RoboDK station: Proyecto-Final.rdk

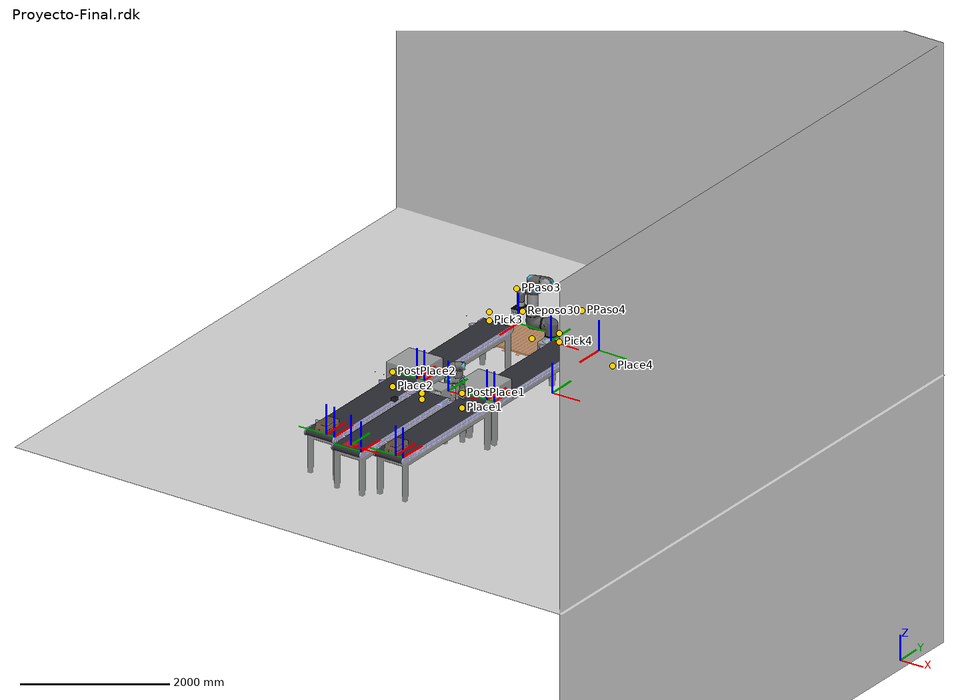
[picture v0: the station drawn from its stored meshes, robots at their saved joint values, targets as dots, program paths as lines]
Station Proyecto final (saved by RoboDK 6.0.0). Poses are relative to the parent item; angles as X-Y-Z fixed-axis rotations.
Station parameters (name, value as stored): SenyalSensor1, 1, SenyalSensor2, 1, SenyalSensorA, 0, SenyalSensor3, 0, SenyalSensor4, 0, x1, 0, z1, 1, x2, 0, z2, 0, x3, 1.0, y3, 0.0, z3, 0.0, x4, 1.0, y4, 0.0, z4, 0.0, Done1, 0, Done2, 0, LuzPalet1, 0, LuzPalet2, 0, IDAzulejo, 23, Lote1, 1, Lote2, 2, ColaAzulejos, 1, Box-Spawner-Settings-4, Box-Spawner-Settings-4-Backup, Box-Spawner-Settings-0, Box-Spawner-Settings-0-Backup, Box-Spawner-Settings-1, Box-Spawner-Settings-1-Backup
  - frame general at (0, -573.6, 0) mm
    - object Wall1 at (3270, -50, -100) mm, rotated rx 0 ry 90 rz 0 deg, size 8910 x 8910 x 0 mm, geometry from Floor.sld
    - object Wall2 at (-1170, 4410, -100) mm, rotated rx 0 ry 90 rz -90 deg, size 8910 x 8910 x 0 mm, geometry from Floor.sld
    - frame UR5e Base at (-1166.19, -738.6, 0) mm
      - robot UR5e: 6 axes, payload 5 kg, reach 850 mm, repeatability 0.03 mm, weight 18.4 kg
          modified DH rows (alpha deg, a mm, theta deg, d mm): 0, 0, 0, 162.5; 90, 0, 180, 0; 0, 425, 0, 0; 0, 392.25, 0, 133.3; -90, 0, 0, 99.7; 90, 0, 180, 99.6
          joint limits [-360, -360, -360, -360, -360, -360] to [360, 360, 360, 360, 360, 360]; home [0, -90, -90, 0, 90, 0]; saved at [128.528, -52.006, 56.851, -94.846, 269.999, -51.472]
        - tool SMC ZXP7A01-ZP20U-X1 Vacuum Gripper, TCP at (0, 0, 125) mm, size 88 x 106.8 x 127.9 mm
    - frame UR30 Base at (-1166.19, 1647.35, -216.33) mm
      - robot UR30: 6 axes
          modified DH rows (alpha deg, a mm, theta deg, d mm): 0, 0, 0, 236.3; 90, 0, 180, 0; 0, 637, 0, 0; 0, 503.7, 0, 201; -90, 0, 0, 159.3; 90, 0, 180, 150
          joint limits [-360, -360, -360, -360, -360, -360] to [360, 360, 360, 360, 360, 360]; home [0, -90, -90, 0, 90, 0]; saved at [-73.932, -91.682, -77.512, -100.814, -269.956, 16.068]
        - tool OnRobot VGP20 Vacuum Gripper, TCP at (-28.8, 0, 85.19) mm, size 214.7 x 147.3 x 83 mm
    - frame Cinta1 at (-372.38, -2930, 100) mm, rotated rx 0 ry 0 rz 90 deg
      - robot Cajas1: 1 axes
          modified DH rows (alpha deg, a mm, theta deg, d mm): 0, 0, 0, 0 linear
          base shift (0, 0, 0) mm, rotated rx 0 ry 90 rz 0 deg
          joint limits [-500000] to [500000]; home [0]; saved at [0]
        - frame CintaCaja1 at (0, 120, 0) mm
          - object cajaA1 at (0, 0, 0) mm, size 193.3 x 289.9 x 121.2 mm, geometry from Box-24x16in-Open.sld
      - object Fotocelula1 at (1900, 0, 0) mm, rotated rx 90 ry 0 rz 90 deg, size 683.3 x 45.2 x 12.5 mm, geometry from SICK-WL4S-Laser-Sensor.sld
      - target Place1 (Cartesian target) at (1686, 221, 9.7) mm, rotated rx -180 ry 0 rz -180 deg; joints [128.527, -47.564, 68.767, -111.204, 269.999, -51.473] of UR5e
      - target PostPlace1 (Cartesian target) at (1686, 221, 226.03) mm, rotated rx 180 ry 0 rz 180 deg; joints [128.527, -51.577, 43.492, -81.916, 269.999, -51.473] of UR5e
    - frame Cinta2 at (-1498.56, -2930, 100) mm, rotated rx 0 ry 0 rz 90 deg
      - robot Cajas2: 1 axes
          modified DH rows (alpha deg, a mm, theta deg, d mm): 0, 0, 0, 0 linear
          base shift (0, 0, 0) mm, rotated rx 0 ry 90 rz 0 deg
          joint limits [-500000] to [500000]; home [0]; saved at [0]
        - frame CintaCaja2 at (0, 120, 0) mm
          - object cajaA2 at (0, 0, 0) mm, size 193.3 x 289.9 x 121.2 mm, geometry from Box-24x16in-Open.sld
      - object Fotocelula2 at (1900, 0, 0) mm, rotated rx 90 ry 0 rz 90 deg, size 683.3 x 45.2 x 12.5 mm, geometry from SICK-WL4S-Laser-Sensor.sld
      - target Place2 (Cartesian target) at (1686, 221, 9.7) mm, rotated rx 180 ry 0 rz 180 deg; joints [32.16, -49.513, 72.223, -112.711, 270.001, -147.84] of UR5e
      - target PostPlace2 (Cartesian target) at (1686, 221, 226.03) mm, rotated rx 180 ry 0 rz 180 deg; joints [32.16, -54.32, 48.04, -83.72, 270.001, -147.84] of UR5e
    - frame Azulejos at (-940.42, -3100.32, 100) mm, rotated rx 0 ry 0 rz 90 deg
      - robot AzulejoAn: 1 axes
          modified DH rows (alpha deg, a mm, theta deg, d mm): 0, 0, 0, 0 linear
          base shift (0, 0, 0) mm, rotated rx 0 ry 90 rz 0 deg
          joint limits [-500000] to [500000]; home [0]; saved at [0]
        - frame CintaAzulejos at (90, 230, 0) mm, rotated rx 0 ry 0 rz -90 deg
          - object Azulejo at (0, 0, 0) mm, size 176.4 x 137.2 x 9.8 mm, geometry from tinker.obj
          - object Azulejo at (0, 0, 0) mm, size 176.4 x 137.2 x 9.8 mm, geometry from tinker.obj
          - object Azulejo at (0, 0, 0) mm, size 176.4 x 137.2 x 9.8 mm, geometry from tinker.obj
          - object Azulejo at (0, 0, 0) mm, size 176.4 x 137.2 x 9.8 mm, geometry from tinker.obj
          - object Azulejo at (0, 0, 0) mm, size 176.4 x 137.2 x 9.8 mm, geometry from tinker.obj
          - object Azulejo at (0, 0, 0) mm, size 176.4 x 137.2 x 9.8 mm, geometry from tinker.obj
          - object Azulejo at (0, 0, 0) mm, size 176.4 x 137.2 x 9.8 mm, geometry from tinker.obj
          - object Azulejo at (0, 0, 0) mm, size 176.4 x 137.2 x 9.8 mm, geometry from tinker.obj
          - object Azulejo at (0, 0, 0) mm, size 176.4 x 137.2 x 9.8 mm, geometry from tinker.obj
          - object Azulejo at (0, 0, 0) mm, size 176.4 x 137.2 x 9.8 mm, geometry from tinker.obj
          - object Azulejo at (0, 0, 0) mm, size 176.4 x 137.2 x 9.8 mm, geometry from tinker.obj
      - object Matrox Iris GTR Camera at (1130, 180, 310) mm, rotated rx 180 ry 0 rz 180 deg, size 76.3 x 92.1 x 55 mm, geometry from Matrox-Iris-GTR-Camera.sld
      - object FotocelulaA at (1850, 0, 0) mm, rotated rx 0 ry 0 rz 90 deg, size 683.3 x 45.2 x 12.5 mm, geometry from SICK-WL4S-Laser-Sensor.sld
      - target Pick (Cartesian target) at (1766.53, 242.5, 8) mm, rotated rx 180 ry 0 rz 180 deg; joints [75.453, -68.071, 102.923, -124.853, 270, -104.547] of UR5e
      - target PrePick (Cartesian target) at (1766.53, 242.5, 95) mm, rotated rx 180 ry 0 rz 180 deg; joints [75.453, -73.796, 96.44, -112.645, 270, -104.547] of UR5e
    - frame Cinta3 at (-1498.56, -835, 100) mm, rotated rx 0 ry 0 rz 90 deg
      - robot Cajas3: 1 axes
          modified DH rows (alpha deg, a mm, theta deg, d mm): 0, 0, 0, 0 linear
          base shift (0, 0, 0) mm, rotated rx 0 ry 90 rz 0 deg
          joint limits [-500000] to [500000]; home [0]; saved at [0]
        - frame CintaCaja3 at (0, 120, 0) mm
          - object cajaC at (0, 0, 0) mm, size 181.1 x 277.6 x 121.7 mm, geometry from Box-24x16in-Closed.sld
          - object cajaC at (0, 0, 0) mm, size 181.1 x 277.6 x 121.7 mm, geometry from Box-24x16in-Closed.sld
      - object Fotocelula3 at (1900, 0, 0) mm, rotated rx 90 ry 0 rz 90 deg, size 683.3 x 45.2 x 12.5 mm, geometry from SICK-WL4S-Laser-Sensor.sld
      - target Pick3 (Cartesian target) at (1780.34, 185.56, 120.53) mm, rotated rx 179.98 ry 0.04 rz 90 deg; joints [-114.864, -111.118, -87.209, -71.708, -269.972, -24.864] of UR30
      - target PrePick3 (Cartesian target) at (1780.34, 185.56, 250.53) mm, rotated rx 179.98 ry 0.04 rz 90 deg; joints [-114.864, -108.804, -75.427, -85.804, -269.972, -24.864] of UR30
    - frame Cinta4 at (-352.38, -835, 100) mm, rotated rx 0 ry 0 rz 90 deg
      - robot Cajas4: 1 axes
          modified DH rows (alpha deg, a mm, theta deg, d mm): 0, 0, 0, 0 linear
          base shift (0, 0, 0) mm, rotated rx 0 ry 90 rz 0 deg
          joint limits [-500000] to [500000]; home [0]; saved at [0]
        - frame CintaCaja4 at (0, 120, 0) mm
          - object cajaC at (0, 0, 0) mm, size 181.1 x 277.6 x 121.7 mm, geometry from Box-24x16in-Closed.sld
          - object cajaC at (0, 0, 0) mm, size 181.1 x 277.6 x 121.7 mm, geometry from Box-24x16in-Closed.sld
      - object Fotocelula4 at (1900, 0, 0) mm, rotated rx 90 ry 0 rz 90 deg, size 683.3 x 45.2 x 12.5 mm, geometry from SICK-WL4S-Laser-Sensor.sld
      - target Pick4 (Cartesian target) at (1780.34, 191.73, 121.32) mm, rotated rx 179.98 ry 0.04 rz 90 deg; joints [-37.962, -112.539, -85.01, -72.432, -269.96, 52.038] of UR30
      - target PrePick4 (Cartesian target) at (1780.34, 191.73, 250.53) mm, rotated rx 179.98 ry 0.04 rz 90 deg; joints [-37.962, -110.369, -73.215, -86.397, -269.96, 52.038] of UR30
    - frame Frame Pallet 1 at (-2170, 2320, -500) mm, rotated rx 0 ry 0 rz -90 deg
      - object Pallet 1130x1130mm at (0, 0, 0) mm, size 706 x 706 x 68.7 mm, geometry from Pallet-1130x1130mm.sld
      - target PPaso3 (Cartesian target) at (739.69, 485.83, 940.76) mm, rotated rx 179.98 ry 0.04 rz -90 deg; joints [-151.611, -76.512, -99.315, -94.218, -269.999, -61.611] of UR30
      - target Place3 (Cartesian target) at (489, 561.4, 120.9) mm, rotated rx 179.98 ry 0.04 rz -90 deg; joints [-177.865, -156.304, -147.246, 33.509, -270.018, -87.865] of UR30
    - frame Frame Pallet 2 at (-812, 2253.67, -500) mm, rotated rx 0 ry 0 rz -90 deg
      - object Pallet 1130x1130mm at (0, 0, 0) mm, size 706 x 706 x 68.7 mm, geometry from Pallet-1130x1130mm.sld
      - target PPaso4 (Cartesian target) at (753.36, 247.81, 965.73) mm, rotated rx 179.98 ry 0.04 rz -90 deg; joints [5.462, -80.617, -93.419, -95.922, -269.984, 95.462] of UR30
      - target Place4 (Cartesian target) at (489, 561.4, 120.9) mm, rotated rx 179.98 ry 0.04 rz -90 deg; joints [-177.865, -156.304, -147.246, 33.509, -270.018, -87.865] of UR30
    - object Mesa4 at (-590, 170, -580) mm, size 465.3 x 1980 x 594 mm, geometry from tinker.obj
    - object Mesa1 at (-590, -1910, -580) mm, size 465.3 x 1980 x 594 mm, geometry from tinker.obj
    - object Mesa2 at (-1720, -1910, -580) mm, size 465.3 x 1980 x 594 mm, geometry from tinker.obj
    - object Mesa3 at (-1720, 170, -580) mm, size 465.3 x 1980 x 594 mm, geometry from tinker.obj
    - object MesaA at (-1160, -2090, -580) mm, size 465.3 x 1980 x 594 mm, geometry from tinker.obj
    - object Soporte30 at (-1166.19, 1647.35, -576.33) mm, size 270 x 270 x 360 mm, geometry from tinker.obj
    - object Soporte5e at (-1166.19, -738.6, -575) mm, size 225 x 225 x 576 mm, geometry from tinker.obj
    - object Tapa1 at (-592, -750, 70) mm, rotated rx 0 ry 0 rz 90 deg, size 540 x 540 x 243 mm, geometry from tinker.obj
    - object Tapa2 at (-1718, -750, 70) mm, rotated rx 0 ry 0 rz 90 deg, size 540 x 540 x 243 mm, geometry from tinker.obj
    - object Basura at (-1158, -950, 60) mm, rotated rx 0 ry 0 rz 90 deg, size 218.7 x 218.7 x 98.4 mm, geometry from tinker.obj
      - object BasuraBajo at (0, 0, 50) mm, rotated rx 180 ry 0 rz 180 deg, size 218.7 x 218.7 x 98.4 mm, geometry from tinker.obj
    - object Floor at (-1140, -50, -570) mm, size 8910 x 8910 x 0 mm, geometry from Floor.sld
    - target Reposo30 (Cartesian target) at (-1144.17, 945.31, 515.93) mm, rotated rx 179.98 ry 0.04 rz 180 deg; joints [-71.585, -90.912, -88.057, -91.037, -269.956, 18.415] of UR30
    - target PuntoPaso1 (Cartesian target) at (-1097.88, -1258.79, 521.04) mm, rotated rx 180 ry 0 rz -90 deg; joints [82.762, -83.23, 58.981, -65.751, 270, -97.238] of UR5e
  - object AzulejoBase at (0, 0, 0) mm, size 176.4 x 137.2 x 9.8 mm, geometry from tinker.obj
  - object cajaBase at (0, 0, 0) mm, size 181.1 x 277.6 x 121.7 mm, geometry from Box-24x16in-Closed.sld
  - program PROGRAMA FINAL (11 instructions, listed below)
  - program RESET TOTAL (7 instructions, listed below)
  - program Set a 0 (17 instructions, listed below)
  - program Set a 0 bd (3 instructions, listed below)
  - folder PROGRAMAS
    - folder Cintas
      - folder Cinta 1
        - Python program ResetCinta1 (listed below)
        - Python program AvanceCinta1 (listed below)
      - folder Cinta 2
        - Python program ResetCinta2 (listed below)
        - Python program AvanceCinta2 (listed below)
      - folder Azulejos
        - Python program ResetCintaA (listed below)
        - Python program AvanceCintaA (listed below)
      - folder Cinta 3
        - Python program ResetCinta3 (listed below)
        - Python program AvanceCinta3 (listed below)
      - folder Cinta 4
        - Python program ResetCinta4 (listed below)
        - Python program AvanceCinta4 (listed below)
    - folder Apilado
      - Python program Apilado (listed below)
    - folder Paletizado
      - Python program Paletizado (listed below)
    - folder Recibe MQTT spawn
      - Python program RobotControllerS (listed below)
      - Python program LeerMQTTS (listed below)
    - folder Recibe MQTT Borrado
      - Python program LeerMQTTB (listed below)
      - Python program RobotControllerB (listed below)
    - folder Envia MQTT
      - Python program FuncioON (listed below)
      - Python program FuncioOFF (listed below)
      - Python program Palet1ON (listed below)
      - Python program Palet1OFF (listed below)
      - Python program Palet2ON (listed below)
      - Python program Palet2OFF (listed below)
    - folder Borrado de Azulejos
      - Python program BorradoAzulejos (listed below)

--- program PROGRAMA FINAL (robot UR5e) ---
  Llamar Set a 0
  Llamar FuncioON
  Ejecutar Paletizado
  Ejecutar AvanceCinta4
  Ejecutar AvanceCinta3
  Ejecutar Apilado
  Ejecutar AvanceCintaA
  Ejecutar AvanceCinta2
  Ejecutar AvanceCinta1
  Ejecutar LeerMQTTB
  Ejecutar LeerMQTTS

--- program RESET TOTAL (robot UR5e) ---
  Llamar FuncioOFF
  Llamar ResetCinta1
  Llamar ResetCinta2
  Llamar ResetCintaA
  Llamar ResetCinta3
  Llamar ResetCinta4
  Llamar BorradoAzulejos

--- program Set a 0 (robot UR5e) ---
  Set SenyalSensor1=0
  Set SenyalSensor2=0
  Set SenyalSensorA=0
  Set SenyalSensor3=0
  Set SenyalSensor4=0
  Set x1=0
  Set z1=0
  Set x2=0
  Set z2=0
  Set x3=0
  Set y3=0
  Set z3=0
  Set x4=0
  Set y4=0
  Set z4=0
  Set Done1=0
  Set Done2=0

--- program Set a 0 bd (robot UR5e) ---
  Set IDAzulejo=0
  Set Lote1=0
  Set Lote2=0

--- Python program ResetCinta1 ---
# Type help("robodk.robolink") or help("robodk.robomath") for more information
# Press F5 to run the script
# Documentation: https://robodk.com/doc/en/RoboDK-API.html
# Reference:     https://robodk.com/doc/en/PythonAPI/robodk.html
# Note: It is not required to keep a copy of this file, your Python script is saved with your RDK project

# You can also use the new version of the API:
from robodk import robolink    # RoboDK API
from robodk import robomath    # Robot toolbox
RDK = robolink.Robolink()

cinta=RDK.Item('Cajas1')

if cinta.Valid():
    cinta.setJoints([0])

--- Python program AvanceCinta1 ---
import time
from robodk import robolink    # RoboDK API
import psycopg

RDK = robolink.Robolink()

caja = RDK.Item('cajaA1')
fotocelula = RDK.Item('Fotocelula1')
frame = RDK.Item('CintaCaja1')
cinta = RDK.Item('Cajas1')
INCREMENTO_MM=406

while(True):
    lista_caja = frame.Childs()
    detectado = False

    while not detectado:
        cinta.MoveJ(cinta.Joints()+INCREMENTO_MM)
        for caja in lista_caja:
            if caja.Name():
                if fotocelula.Collision(caja):
                    detectado = True
                    RDK.setParam('SenyalSensor1', 1)
                    break


    while detectado:
        done = RDK.getParam('Done1')
        if done == 1:
            detectado = False
        time.sleep(0.1)

    conn = psycopg.connect(
            dbname = "Azulejos",
            user = "postgres",
            password = "8130",
            host = "localhost",
            port = "5432"
    )
    cur = conn.cursor()

    lote1 = int(RDK.getParam('Lote1'))
    lote2 = int(RDK.getParam('Lote2'))
    if lote1 == 0 and lote2 == 0:
        lote2 = 1
    elif lote1 > lote2:
        lote2 = lote1 + 1
    else:
        lote2 = lote2 + 1
    lote = f"L-{lote2:03d}"

    sql = """INSERT INTO azulejos.Caja_llena (ID_lote, Tamano, Tipo, Codigo_Compra)
    VALUES (%s, %s, %s, %s)"""
    datos = (lote, 10, 'bueno', f"P25-{lote2:03d}")
    cur.execute(sql, datos)
    conn.commit()

    RDK.setParam('Lote2', lote2)
    cur.close()
    conn.close()

    cinta.MoveJ(cinta.Joints()+INCREMENTO_MM)
    RDK.setParam('SenyalSensor1', 0)
    lista_caja = frame.Childs()

    for item in lista_caja:
        if item.Name().startswith('Azulejo'):
            item.Delete()

    RDK.setParam('Done1', 0)
    cinta.setJoints([0])

--- Python program ResetCinta2 ---
# Type help("robodk.robolink") or help("robodk.robomath") for more information
# Press F5 to run the script
# Documentation: https://robodk.com/doc/en/RoboDK-API.html
# Reference:     https://robodk.com/doc/en/PythonAPI/robodk.html
# Note: It is not required to keep a copy of this file, your Python script is saved with your RDK project

# You can also use the new version of the API:
from robodk import robolink    # RoboDK API
from robodk import robomath    # Robot toolbox
RDK = robolink.Robolink()

cinta=RDK.Item('Cajas2')

if cinta.Valid():
    cinta.setJoints([0])

--- Python program AvanceCinta2 ---
import time
from robodk import robolink    # RoboDK API
import psycopg

RDK = robolink.Robolink()

caja = RDK.Item('cajaA2')
fotocelula = RDK.Item('Fotocelula2')
frame = RDK.Item('CintaCaja2')
cinta = RDK.Item('Cajas2')
INCREMENTO_MM=406

while(True):
    lista_caja = frame.Childs()
    detectado = False

    while not detectado:
        cinta.MoveJ(cinta.Joints()+INCREMENTO_MM)
        for caja in lista_caja:
            if caja.Name():
                if fotocelula.Collision(caja):
                    detectado = True
                    RDK.setParam('SenyalSensor2', 1)
                    break


    while detectado:
        done = RDK.getParam('Done2')
        if done == 1:
            detectado = False
        time.sleep(0.1)

    conn = psycopg.connect(
            dbname = "Azulejos",
            user = "postgres",
            password = "8130",
            host = "localhost",
            port = "5432"
    )
    cur = conn.cursor()

    lote1 = int(RDK.getParam('Lote1'))
    lote2 = int(RDK.getParam('Lote2'))
    if lote1 == 0 and lote2 == 0:
        lote1 = 1
    elif lote1 > lote2:
        lote1 = lote1 + 1
    else:
        lote1 = lote2 + 1
    lote = f"L-{lote1:03d}"

    sql = """INSERT INTO azulejos.Caja_llena (ID_lote, Tamano, Tipo, Codigo_Compra)
    VALUES (%s, %s, %s, %s)"""
    datos = (lote, 10, 'defectuoso', f"P25-{lote1:03d}")
    cur.execute(sql, datos)
    conn.commit()

    RDK.setParam('Lote1', lote1)
    cur.close()
    conn.close()

    cinta.MoveJ(cinta.Joints()+INCREMENTO_MM)
    RDK.setParam('SenyalSensor2', 0)
    lista_caja = frame.Childs()

    for item in lista_caja:
        if item.Name().startswith('Azulejo'):
            item.Delete()

    RDK.setParam('Done2', 0)
    cinta.setJoints([0])

--- Python program ResetCintaA ---
# Type help("robodk.robolink") or help("robodk.robomath") for more information
# Press F5 to run the script
# Documentation: https://robodk.com/doc/en/RoboDK-API.html
# Reference:     https://robodk.com/doc/en/PythonAPI/robodk.html
# Note: It is not required to keep a copy of this file, your Python script is saved with your RDK project

# You can also use the new version of the API:
from robodk import robolink    # RoboDK API
from robodk import robomath    # Robot toolbox
RDK = robolink.Robolink()

cinta = RDK.Item('AzulejoAn')

if cinta.Valid():
    cinta.setJoints([0])

--- Python program AvanceCintaA ---
import time
from robodk import robolink    # RoboDK API
from robodk import robomath

RDK = robolink.Robolink()

azulejo = RDK.Item('Azulejo')
fotocelula = RDK.Item('FotocelulaA')
frame = RDK.Item('CintaAzulejos')
cinta = RDK.Item('AzulejoAn')
INCREMENTO_MM = 1680
INCREMENTO_B = 350
lista_azulejos = frame.Childs()
tipo = RDK.getParam('TipoAzulejo')

def spawnear_azulejo():

    template = RDK.Item('AzulejoBase')

    if not template.Valid():
        print("Error: No encuentro el template")
        return None

    template.Copy()
    nuevo_azulejo = RDK.Paste(frame)
    nuevo_azulejo.setName("Azulejo")
    nuevo_azulejo.setVisible(True)
    nuevo_azulejo.setPose(robomath.eye(4))

    return nuevo_azulejo


while(True):
    lista_azulejos = frame.Childs()
    detectado = False

    while not detectado:
        cinta.MoveJ(cinta.Joints()+INCREMENTO_MM)
        for azulejo in lista_azulejos:
            if azulejo.Name().startswith("Azulejo"):
                if fotocelula.Collision(azulejo):
                    detectado = True
                    RDK.setParam('SenyalSensorA', 1)
                    break

    while detectado:
        for azulejo in lista_azulejos:
            if azulejo.Name().startswith("Azulejo"):
                if not fotocelula.Collision(azulejo):
                    detectado = False
                    RDK.setParam('SenyalSensorA', 0)
                    break

    time.sleep(1)

    cinta.setJoints([0])
    azulejo = spawnear_azulejo()

--- Python program ResetCinta3 ---
# Type help("robodk.robolink") or help("robodk.robomath") for more information
# Press F5 to run the script
# Documentation: https://robodk.com/doc/en/RoboDK-API.html
# Reference:     https://robodk.com/doc/en/PythonAPI/robodk.html
# Note: It is not required to keep a copy of this file, your Python script is saved with your RDK project

# You can also use the new version of the API:
from robodk import robolink    # RoboDK API
from robodk import robomath    # Robot toolbox
RDK = robolink.Robolink()

cinta=RDK.Item('Cajas3')

if cinta.Valid():
    cinta.setJoints([0])

--- Python program AvanceCinta3 ---
import time
from robodk import robolink    # RoboDK API
from robodk import robomath

RDK = robolink.Robolink()

caja = RDK.Item('cajaC')
fotocelula = RDK.Item('Fotocelula3')
frame = RDK.Item('CintaCaja3')
cinta = RDK.Item('Cajas3')
INCREMENTO_MM=406

def spawnear_caja():

    template = RDK.Item('cajaBase')

    if not template.Valid():
        print("Error: No encuentro el template")
        return None

    template.Copy()
    nueva_caja = RDK.Paste(frame)
    nueva_caja.setName("cajaC")
    nueva_caja.setVisible(True)
    nueva_caja.setPose(robomath.eye(4))

    return nueva_caja

while(True):
    lista_caja = frame.Childs()
    detectado = False
    Done = RDK.getParam('Done2')

    if Done == 1:
        time.sleep(1)
        while not detectado:
            cinta.MoveJ(cinta.Joints()+INCREMENTO_MM)
            for caja in lista_caja:
                if caja.Name().startswith("cajaC"):
                    if fotocelula.Collision(caja):
                        detectado = True
                        RDK.setParam('SenyalSensor3', 1)
                        break

        while detectado:
            for caja in lista_caja:
                if caja.Name().startswith("cajaC"):
                    if not fotocelula.Collision(caja):
                        detectado = False
                        RDK.setParam('SenyalSensor3', 0)
                        break
            time.sleep(0.1)

        cinta.setJoints([0])
        caja = spawnear_caja()

--- Python program ResetCinta4 ---
# Type help("robodk.robolink") or help("robodk.robomath") for more information
# Press F5 to run the script
# Documentation: https://robodk.com/doc/en/RoboDK-API.html
# Reference:     https://robodk.com/doc/en/PythonAPI/robodk.html
# Note: It is not required to keep a copy of this file, your Python script is saved with your RDK project

# You can also use the new version of the API:
from robodk import robolink    # RoboDK API
from robodk import robomath    # Robot toolbox
RDK = robolink.Robolink()

cinta=RDK.Item('Cajas4')

if cinta.Valid():
    cinta.setJoints([0])

--- Python program AvanceCinta4 ---
import time
from robodk import robolink    # RoboDK API
from robodk import robomath

RDK = robolink.Robolink()

caja = RDK.Item('cajaC')
fotocelula = RDK.Item('Fotocelula4')
frame = RDK.Item('CintaCaja4')
cinta = RDK.Item('Cajas4')
INCREMENTO_MM=406

def spawnear_caja():

    template = RDK.Item('cajaBase')

    if not template.Valid():
        print("Error: No encuentro el template")
        return None

    template.Copy()
    nueva_caja = RDK.Paste(frame)
    nueva_caja.setName("cajaC")
    nueva_caja.setVisible(True)
    nueva_caja.setPose(robomath.eye(4))

    return nueva_caja

while(True):
    lista_caja = frame.Childs()
    detectado = False
    Done = RDK.getParam('Done1')

    if Done == 1:
        time.sleep(1)
        while not detectado:
            cinta.MoveJ(cinta.Joints()+INCREMENTO_MM)
            for caja in lista_caja:
                if caja.Name().startswith("cajaC"):
                    if fotocelula.Collision(caja):
                        detectado = True
                        RDK.setParam('SenyalSensor4', 1)
                        break

        while detectado:
            for caja in lista_caja:
                if caja.Name().startswith("cajaC"):
                    if not fotocelula.Collision(caja):
                        detectado = False
                        RDK.setParam('SenyalSensor4', 0)
                        break
            time.sleep(0.1)

        cinta.setJoints([0])
        caja = spawnear_caja()

--- Python program Apilado ---
# Type help("robodk.robolink") or help("robodk.robomath") for more information
# Press F5 to run the script
# Documentation: https://robodk.com/doc/en/RoboDK-API.html
# Reference:     https://robodk.com/doc/en/PythonAPI/robodk.html
# Note: It is not required to keep a copy of this file, your Python script is saved with your RDK project
import time
from robodk import robolink    # RoboDK API
from robodk import robomath    # Robot toolbox
import psycopg

RDK = robolink.Robolink()

conn = psycopg.connect(
    dbname = "Azulejos",
    user = "postgres",
    password = "8130",
    host = "localhost",
    port = "5432"
)
cur = conn.cursor()

#TIPO 3

INCREMENTO_B = 350
cinta = RDK.Item('AzulejoAn')
frame = RDK.Item('CintaAzulejos')
lista_azulejos = frame.Childs()

#ROBOT
robot = RDK.Item('UR5e', robolink.ITEM_TYPE_ROBOT)

#TARGETS
target_PPaso = RDK.Item('PuntoPaso1', robolink.ITEM_TYPE_TARGET)
target_Pick = RDK.Item('Pick', robolink.ITEM_TYPE_TARGET)
target_PrePick = RDK.Item('PrePick', robolink.ITEM_TYPE_TARGET)
target_Place1 = RDK.Item('Place1', robolink.ITEM_TYPE_TARGET)
target_Place2 = RDK.Item('Place2', robolink.ITEM_TYPE_TARGET)
target_PostPlace1 = RDK.Item('PostPlace1', robolink.ITEM_TYPE_TARGET)
target_PostPlace2 = RDK.Item('PostPlace2', robolink.ITEM_TYPE_TARGET)

#OBJETOS
azulejo = RDK.Item('Azulejo', robolink.ITEM_TYPE_OBJECT)

#HERRAMIENTA
ventosa = RDK.Item('SMC ZXP7A01-ZP20U-X1 Vacuum Gripper', robolink.ITEM_TYPE_TOOL)

#FRAMES
general = RDK.Item('general', robolink.ITEM_TYPE_FRAME)
frameCintaA = RDK.Item('Azulejos', robolink.ITEM_TYPE_FRAME)
frameAzulejo = RDK.Item('CintaAzulejos', robolink.ITEM_TYPE_FRAME)
frameCinta1 = RDK.Item('Cinta1', robolink.ITEM_TYPE_FRAME)
frameCinta2 = RDK.Item('Cinta2', robolink.ITEM_TYPE_FRAME)
frameCaja1 = RDK.Item('CintaCaja1', robolink.ITEM_TYPE_FRAME)
frameCaja2 = RDK.Item('CintaCaja2', robolink.ITEM_TYPE_FRAME)

target_PPaso.setParent(general)
target_Pick.setParent(frameCintaA)
target_PrePick.setParent(frameCintaA)
target_Place1.setParent(frameCinta1)
target_Place2.setParent(frameCinta2)
target_PostPlace1.setParent(frameCinta1)
target_PostPlace2.setParent(frameCinta2)

def formatear_serie(numero_serie):
    bloque_serie = ((numero_serie - 1) // 999) + 1
    numero_en_bloque = ((numero_serie - 1) % 999) + 1
    return f"S{bloque_serie}-{numero_en_bloque:03d}"

# --- CÓDIGO PRINCIPAL ---

while(True):
    cola_raw = RDK.getParam('ColaAzulejos')

    if isinstance(cola_raw, (float, int)):
        cola_actual = str(int(cola_raw))
    elif cola_raw:
        cola_actual = str(cola_raw)
    else:
        cola_actual = ""

    try:
        SensorA = int(RDK.getParam('SenyalSensorA'))
    except:
        SensorA = 0

    if SensorA == 1 and cola_actual:

        lista_ordenes = cola_actual.split(',')

        try:
            tipo_actual = int(lista_ordenes[0])
        except ValueError:
            tipo_actual = 0

        if lista_ordenes[1:] == []:
            RDK.setParam('ColaAzulejos',1)
        else:
            elementos_restantes = lista_ordenes[1:]
            RDK.setParam('ColaAzulejos', ",".join(elementos_restantes))

        #GDI

        lote1 = int(RDK.getParam('Lote1'))
        lote2 = int(RDK.getParam('Lote2'))
        lote_aux = 0
        estado = 0

        if tipo_actual == 1:
            estado = 'bueno'
            lote_aux = lote2
        elif tipo_actual == 2:
            estado = 'defectuoso'
            lote_aux = lote1
        elif tipo_actual == 3:
            estado = 'roto'
            lote = 'Basura'

        ID = int(RDK.getParam('IDAzulejo'))

        numero_serie = ID + 1
        serie = formatear_serie(numero_serie)
        if tipo_actual == 1 or tipo_actual == 2:
            lote = f"L-{lote_aux:03d}"

        sql = """INSERT INTO azulejos.Azulejo (N_serie, Estado, ID_lote)
        VALUES (%s, %s, %s)"""
        datos = (serie, estado, lote)
        cur.execute(sql, datos)
        conn.commit()
        RDK.setParam('IDAzulejo', numero_serie)

        if tipo_actual != 3:

            # PICK
            robot.setPoseFrame(general)
            robot.setSpeed(500,100)
            robot.MoveJ(target_PPaso.Pose())

            robot.setPoseFrame(frameCintaA)
            robot.MoveJ(target_PrePick.Pose())
            robot.MoveL(target_Pick.Pose())

            azulejos_disponibles = frameAzulejo.Childs()

            if len(azulejos_disponibles) > 0:
                azulejo_actual = azulejos_disponibles[0]
                azulejo_actual.setParentStatic(ventosa)

            robot.MoveL(target_PrePick.Pose())

            match tipo_actual:

                case 1:
                    time.sleep(1)
                    while int(RDK.getParam('SenyalSensor1')) != 1:
                        time.sleep(0.1)

                    robot.setPoseFrame(general)
                    robot.setSpeed(500,100)
                    robot.MoveJ(target_PPaso.Pose())

                    try:
                        x1 = int(RDK.getParam('x1'))
                        z1 = int(RDK.getParam('z1'))
                    except:
                        x1, z1 = 0, 0

                    desplazamiento1 = robomath.transl(x1*-137, 0, z1*-10)
                    pose_place1 = target_Place1.Pose() * desplazamiento1

                    # Place1
                    robot.setPoseFrame(frameCinta1)
                    robot.MoveL(pose_place1 * robomath.transl([0,0,-120]))
                    robot.setSpeed(50,20)
                    robot.MoveL(pose_place1)
                    time.sleep(1)
                    azulejo_actual.setParentStatic(frameCaja1)

                    robot.setPoseFrame(frameCinta1)
                    robot.setSpeed(500,100)
                    robot.MoveL(target_PostPlace1.Pose())

                    robot.setPoseFrame(general)
                    robot.setSpeed(500,100)
                    robot.MoveJ(target_PPaso.Pose())

                    if x1 < 2:
                        x1 = x1 + 1
                    if x1 == 2:
                        z1 = z1 + 1
                        x1 = 0
                    if z1 == 5:
                        x1 = 0
                        z1 = 0
                        RDK.setParam('Done1', 1)
                        time.sleep(2)

                    RDK.setParam('x1', str(x1))
                    RDK.setParam('z1', str(z1))

                case 2:
                    time.sleep(1)
                    while int(RDK.getParam('SenyalSensor2')) != 1:
                        time.sleep(0.1)

                    robot.setPoseFrame(general)
                    robot.setSpeed(500,100)
                    robot.MoveJ(target_PPaso.Pose())

                    try:
                        x2 = int(RDK.getParam('x2'))
                        z2 = int(RDK.getParam('z2'))
                    except:
                        x2, z2 = 0, 0

                    desplazamiento2 = robomath.transl(x2*-137, 0, z2*-10)
                    pose_place2 = target_Place2.Pose() * desplazamiento2

                    # Place2
                    robot.setPoseFrame(frameCinta2)
                    robot.MoveL(pose_place2 * robomath.transl([0,0,-120]))
                    robot.setSpeed(50,20)
                    robot.MoveL(pose_place2)
                    time.sleep(1)
                    azulejo_actual.setParentStatic(frameCaja2)

                    robot.setPoseFrame(frameCinta2)
                    robot.setSpeed(500,100)
                    robot.MoveL(target_PostPlace2.Pose())

                    robot.setPoseFrame(general)
                    robot.setSpeed(500,100)
                    robot.MoveJ(target_PPaso.Pose())

                    if x2 < 2:
                        x2 = x2 + 1
                    if x2 == 2:
                        z2 = z2 + 1
                        x2 = 0
                    if z2 == 5:
                        x2 = 0
                        z2 = 0
                        RDK.setParam('Done2', 1)

                    RDK.setParam('x2', str(x2))
                    RDK.setParam('z2', str(z2))
        elif tipo_actual == 3:
            cinta.MoveJ(cinta.Joints() + INCREMENTO_B)
            for item in lista_azulejos:
                if item.Valid() and item.Name().startswith('Azulejo'):
                    item.Delete()
                    lista_azulejos.remove(item)
                    break

    else:
        time.sleep(0.1)

cur.close()
conn.close()

--- Python program Paletizado ---
# Type help("robodk.robolink") or help("robodk.robomath") for more information
# Press F5 to run the script
# Documentation: https://robodk.com/doc/en/RoboDK-API.html
# Reference:     https://robodk.com/doc/en/PythonAPI/robodk.html
# Note: It is not required to keep a copy of this file, your Python script is saved with your RDK project

# You can also use the new version of the API:
import time
from robodk import robolink    # RoboDK API
from robodk import robomath    # Robot toolbox
RDK = robolink.Robolink()

#ROBOT

robot = RDK.Item('UR30', robolink.ITEM_TYPE_ROBOT)

#PROGRAMAS

prog1 = RDK.Item('Palet1ON')
prog2 = RDK.Item('Palet2ON')

#TARGETS

target_Reposo = RDK.Item('Reposo30', robolink.ITEM_TYPE_TARGET)
target_PPaso1 = RDK.Item('PPaso3', robolink.ITEM_TYPE_TARGET)
target_PPaso2 = RDK.Item('PPaso4', robolink.ITEM_TYPE_TARGET)
target_Pick1 = RDK.Item('Pick3', robolink.ITEM_TYPE_TARGET)
target_PrePick1 = RDK.Item('PrePick3', robolink.ITEM_TYPE_TARGET)
target_Pick2 = RDK.Item('Pick4', robolink.ITEM_TYPE_TARGET)
target_PrePick2 = RDK.Item('PrePick4', robolink.ITEM_TYPE_TARGET)
target_Place1 = RDK.Item('Place3', robolink.ITEM_TYPE_TARGET)
target_Place2 = RDK.Item('Place4', robolink.ITEM_TYPE_TARGET)

#OBJETOS

caja = RDK.Item('cajaC', robolink.ITEM_TYPE_OBJECT)

#HERRAMIENTA

ventosa = RDK.Item('OnRobot VGP20 Vacuum Gripper', robolink.ITEM_TYPE_TOOL)

#FRAMES

general = RDK.Item('general', robolink.ITEM_TYPE_FRAME)
frameCinta3 = RDK.Item('Cinta3', robolink.ITEM_TYPE_FRAME)
frameCinta4 = RDK.Item('Cinta4', robolink.ITEM_TYPE_FRAME)
frameCintaCaja3 = RDK.Item('CintaCaja3', robolink.ITEM_TYPE_FRAME)
frameCintaCaja4 = RDK.Item('CintaCaja4', robolink.ITEM_TYPE_FRAME)
framePalet1 = RDK.Item('Frame Pallet 1', robolink.ITEM_TYPE_FRAME)
framePalet2 = RDK.Item('Frame Pallet 2', robolink.ITEM_TYPE_FRAME)

target_Reposo.setParent(general)
target_PPaso1.setParent(framePalet1)
target_PPaso2.setParent(framePalet2)
target_Pick1.setParent(frameCinta3)
target_PrePick1.setParent(frameCinta3)
target_Pick2.setParent(frameCinta4)
target_PrePick2.setParent(frameCinta4)
target_Place1.setParent(framePalet1)
target_Place2.setParent(framePalet2)

#CÓDIGO

while(True):
    tipo = 0
    while int(RDK.getParam('SenyalSensor4')) != 1 and int(RDK.getParam('SenyalSensor3')) != 1:
        time.sleep(0.1)
    if int(RDK.getParam('SenyalSensor4')) == 1:
        tipo = 2
    elif int(RDK.getParam('SenyalSensor3')) == 1:
        tipo = 1

    match tipo:

        case 1:

            #PICK

            if int(RDK.getParam('LuzPalet1')) == 0:

                robot.setPoseFrame(general)
                robot.setSpeed(500,100)
                robot.MoveJ(target_Reposo.Pose())

                robot.setPoseFrame(frameCinta3)
                robot.MoveJ(target_PrePick1.Pose())
                robot.MoveL(target_Pick1.Pose())

                caja_disponible = frameCintaCaja3.Childs()

                if len(caja_disponible) > 0:

                    caja_actual = caja_disponible[0]
                    caja_actual.setParentStatic(ventosa)

                robot.MoveL(target_PrePick1.Pose())

                robot.setPoseFrame(framePalet1)
                robot.setSpeed(500,100)
                robot.MoveJ(target_PPaso1.Pose())

                x3 = RDK.getParam('x3')
                y3 = RDK.getParam('y3')
                z3 = RDK.getParam('z3')
                luz1 = 0

                desplazamiento1 = robomath.transl(x3*180, y3*280, z3*-120)

                pose_place1 = target_Place1.Pose() * desplazamiento1

                #Place

                robot.MoveL(pose_place1 * robomath.transl([0,0,-120]))
                robot.setSpeed(50,20)
                robot.MoveL(pose_place1)
                time.sleep(1)
                caja_actual.setParentStatic(framePalet1)
                robot.setSpeed(500,100)
                robot.MoveL(target_PPaso1.Pose())

                if x3 < 3:
                    x3 = x3 + 1
                if x3 == 3:
                    y3 = y3 + 1
                    x3 = 0
                if y3 == 2:
                    x3 = 0
                    y3 = 0
                    z3 = z3 + 1
                if z3 == 3:
                    prog1.RunProgram()
                    luz1 = 1
                    x3 = 0
                    y3 = 0
                    z3 = 0

                RDK.setParam('x3',x3)
                RDK.setParam('y3',y3)
                RDK.setParam('z3',z3)
                RDK.setParam('LuzPalet1',luz1)

                robot.setPoseFrame(general)
                robot.setSpeed(500,100)
                robot.MoveJ(target_Reposo.Pose())

        case 2:

            #PICK

            if int(RDK.getParam('LuzPalet2')) == 0:

                robot.setPoseFrame(general)
                robot.setSpeed(500,100)
                robot.MoveJ(target_Reposo.Pose())

                robot.setPoseFrame(frameCinta4)
                robot.MoveJ(target_PrePick2.Pose())
                robot.MoveL(target_Pick2.Pose())

                caja_disponible = frameCintaCaja4.Childs()

                if len(caja_disponible) > 0:

                    caja_actual = caja_disponible[0]
                    caja_actual.setParentStatic(ventosa)

                robot.MoveL(target_PrePick2.Pose())

                robot.setPoseFrame(framePalet2)
                robot.setSpeed(500,100)
                robot.MoveJ(target_PPaso2.Pose())

                x4 = RDK.getParam('x4')
                y4 = RDK.getParam('y4')
                z4 = RDK.getParam('z4')
                luz2 = 0

                desplazamiento2 = robomath.transl(x4*180, y4*280, z4*-120)

                pose_place2 = target_Place2.Pose() * desplazamiento2

                #Place

                robot.MoveL(pose_place2 * robomath.transl([0,0,-120]))
                robot.setSpeed(50,20)
                robot.MoveL(pose_place2)
                time.sleep(1)
                caja_actual.setParentStatic(framePalet2)
                robot.setSpeed(500,100)
                robot.MoveL(target_PPaso2.Pose())

                if x4 < 3:
                    x4 = x4 + 1
                if x4 == 3:
                    y4 = y4 + 1
                    x4 = 0
                if y4 == 2:
                    x4 = 0
                    y4 = 0
                    z4 = z4 + 1
                if z4 == 3:
                    prog2.RunProgram()
                    luz2 = 1
                    x4 = 0
                    y4 = 0
                    z4 = 0

                RDK.setParam('x4',x4)
                RDK.setParam('y4',y4)
                RDK.setParam('z4',z4)
                RDK.setParam('LuzPalet2',luz2)

                robot.setPoseFrame(general)
                robot.setSpeed(500,100)
                robot.MoveJ(target_Reposo.Pose())

--- Python program RobotControllerS ---
# Contenido de RobotController.py

def handle_message(mqtt_client, topic, mensaje, RDK):

    # 1. Convertimos el mensaje a un número
    try:
        tipo = int(mensaje)
    except ValueError:
        print(f"Error: El mensaje '{mensaje}' no es un número. Ignorando orden.")
        return


    cola_raw = RDK.getParam('ColaAzulejos')

    if isinstance(cola_raw, (float, int)):
        cola_actual = str(int(cola_raw))
    elif cola_raw:
        cola_actual = str(cola_raw)
    else:
        cola_actual = ""


    if not cola_actual:
        RDK.setParam('ColaAzulejos', str(tipo))

    else:
        nueva_cola = cola_actual + "," + str(tipo)
        RDK.setParam('ColaAzulejos', nueva_cola)

--- Python program LeerMQTTS ---
from robodk import robolink    # RoboDK API
from robodk import robomath    # Robot toolbox
RDK = robolink.Robolink()

import paho.mqtt.client as mqtt
import RobotControllerS as rc


broker="broker.emqx.io"
port=1883
#user="giirob"
#passwd="UPV2024"
base_topic="sim/working/button/spawn"
#station_name="/demo"
#station_commands_topic=base_topic+station_name+"/commands"
#station_status_topic=base_topic+station_name+"/status"


def on_message(mqttc, obj, msg):
    payload = msg.payload.decode('utf-8')
    topic = msg.topic
    qos = msg.qos
    rc.handle_message(mqttc, topic, payload, RDK)

mqttc = mqtt.Client(mqtt.CallbackAPIVersion.VERSION2)
mqttc.on_message = on_message

#mqttc.username_pw_set(username=user, password=passwd)
mqttc.connect(broker, port, 60)
mqttc.subscribe(base_topic, 0)

mqttc.publish(base_topic, "ready")

mqttc.loop_forever()

--- Python program LeerMQTTB ---
from robodk import robolink    # RoboDK API
from robodk import robomath    # Robot toolbox
import sys                     # Librería del sistema de Python

RDK = robolink.Robolink()

# 1. Le preguntamos a RoboDK en qué carpeta de Windows está guardado el archivo .rdk (tu GitHub)
carpeta_estacion = RDK.getParam('PATH_OPENSTATION')

# 2. Le decimos a Python que añada esa carpeta a su radar de búsqueda
if carpeta_estacion not in sys.path:
    sys.path.append(carpeta_estacion)

import paho.mqtt.client as mqtt
import RobotControllerB as rc


broker="broker.emqx.io"
port=1883
#user="giirob"
#passwd="UPV2024"
base_topic="sim/working/button/empty"
#station_name="/demo"
#station_commands_topic=base_topic+station_name+"/commands"
#station_status_topic=base_topic+station_name+"/status"


def on_message(mqttc, obj, msg):
    payload = msg.payload.decode('utf-8')
    topic = msg.topic
    qos = msg.qos
    rc.handle_message(mqttc, topic, payload, RDK)

mqttc = mqtt.Client(mqtt.CallbackAPIVersion.VERSION2)
mqttc.on_message = on_message

#mqttc.username_pw_set(username=user, password=passwd)
mqttc.connect(broker, port, 60)
mqttc.subscribe(base_topic, 0)

mqttc.publish(base_topic, "ready")

mqttc.loop_forever()

--- Python program RobotControllerB ---
# Contenido de RobotController.py

def handle_message(mqtt_client, topic, mensaje, RDK):
    print(f"--> Nuevo mensaje en {topic}: {mensaje}")

    try:
        tipo = int(mensaje)
    except ValueError:
        print(f"Error: El mensaje '{mensaje}' no es un número. Ignorando orden.")
        return

    # ¡Líneas de robolink eliminadas! Usamos el RDK que viene por los parámetros.

    prog1 = RDK.Item('Palet1OFF')
    prog2 = RDK.Item('Palet2OFF')

    frame1 = RDK.Item('Frame Pallet 1')
    frame2 = RDK.Item('Frame Pallet 2')

    lista_palet1 = frame1.Childs()
    lista_palet2 = frame2.Childs()

    match tipo:
        case 1:
            # 1. Comprobamos que el programa existe para evitar fallos
            if not prog1.Valid():
                print("Error: No se encontró el programa 'Palet1OFF'")
                return

            for item in lista_palet1:
                # Buena práctica: Validar antes de leer el nombre (como vimos antes)
                if item.Valid() and item.Name().startswith('cajaC'):
                    item.Delete()

            RDK.setParam('x3', 0)
            RDK.setParam('y3', 0)
            RDK.setParam('z3', 0)
            RDK.setParam('LuzPalet1', 0)

            # 2. Ejecutamos e imprimimos el resultado
            resultado = prog1.RunProgram()
            if resultado == 0:
                print("Éxito: Programa Palet1OFF iniciado.")
            else:
                print("Fallo: RoboDK rechazó iniciar el programa. (¿El robot está ocupado?)")

        case 2:
            if not prog2.Valid():
                print("Error: No se encontró el programa 'Palet2OFF'")
                return

            for item in lista_palet2:
                if item.Valid() and item.Name().startswith('cajaC'):
                    item.Delete()

            RDK.setParam('x4', 0)
            RDK.setParam('y4', 0)
            RDK.setParam('z4', 0)
            RDK.setParam('LuzPalet2', 0)

            prog2.RunProgram()

--- Python program FuncioON ---
# Ejemplo de un nuevo programa: enviar_alerta.py
import paho.mqtt.client as mqtt

# 1. Configuración
broker = "broker.emqx.io"
port = 1883
# user = "giirob"
# passwd = "UPV2024"
topic_destino = "sim/working"

# 2. Conexión rápida
mqttc = mqtt.Client(mqtt.CallbackAPIVersion.VERSION2)
#mqttc.username_pw_set(username=user, password=passwd)
mqttc.connect(broker, port, 60)

# 3. ¡Disparar el mensaje!
mensaje = "on"
mqttc.publish(topic_destino, mensaje)

# 4. Desconectar (Es buena práctica si el script termina aquí)
mqttc.disconnect()

--- Python program FuncioOFF ---
# Ejemplo de un nuevo programa: enviar_alerta.py
import paho.mqtt.client as mqtt

# 1. Configuración
broker = "broker.emqx.io"
port = 1883
# user = "giirob"
# passwd = "UPV2024"
topic_destino = "sim/working"

# 2. Conexión rápida
mqttc = mqtt.Client(mqtt.CallbackAPIVersion.VERSION2)
#mqttc.username_pw_set(username=user, password=passwd)
mqttc.connect(broker, port, 60)

# 3. ¡Disparar el mensaje!
mensaje = "off"
mqttc.publish(topic_destino, mensaje)

# 4. Desconectar (Es buena práctica si el script termina aquí)
mqttc.disconnect()

--- Python program Palet1ON ---
# Ejemplo de un nuevo programa: enviar_alerta.py
import paho.mqtt.client as mqtt

# 1. Configuración
broker = "broker.emqx.io"
port = 1883
# user = "giirob"
# passwd = "UPV2024"
topic_destino = "sim/working/palet1"

# 2. Conexión rápida
mqttc = mqtt.Client(mqtt.CallbackAPIVersion.VERSION2)
#mqttc.username_pw_set(username=user, password=passwd)
mqttc.connect(broker, port, 60)

# 3. ¡Disparar el mensaje!
mensaje = "on"
mqttc.publish(topic_destino, mensaje)

# 4. Desconectar (Es buena práctica si el script termina aquí)
mqttc.disconnect()

--- Python program Palet1OFF ---
# Ejemplo de un nuevo programa: enviar_alerta.py
import paho.mqtt.client as mqtt

# 1. Configuración
broker = "broker.emqx.io"
port = 1883
# user = "giirob"
# passwd = "UPV2024"
topic_destino = "sim/working/palet1"

# 2. Conexión rápida
mqttc = mqtt.Client(mqtt.CallbackAPIVersion.VERSION2)
#mqttc.username_pw_set(username=user, password=passwd)
mqttc.connect(broker, port, 60)

# 3. ¡Disparar el mensaje!
mensaje = "off"
mqttc.publish(topic_destino, mensaje)

# 4. Desconectar (Es buena práctica si el script termina aquí)
mqttc.disconnect()

--- Python program Palet2ON ---
# Ejemplo de un nuevo programa: enviar_alerta.py
import paho.mqtt.client as mqtt

# 1. Configuración
broker = "broker.emqx.io"
port = 1883
# user = "giirob"
# passwd = "UPV2024"
topic_destino = "sim/working/palet2"

# 2. Conexión rápida
mqttc = mqtt.Client(mqtt.CallbackAPIVersion.VERSION2)
#mqttc.username_pw_set(username=user, password=passwd)
mqttc.connect(broker, port, 60)

# 3. ¡Disparar el mensaje!
mensaje = "on"
mqttc.publish(topic_destino, mensaje)

# 4. Desconectar (Es buena práctica si el script termina aquí)
mqttc.disconnect()

--- Python program Palet2OFF ---
# Ejemplo de un nuevo programa: enviar_alerta.py
import paho.mqtt.client as mqtt

# 1. Configuración
broker = "broker.emqx.io"
port = 1883
# user = "giirob"
# passwd = "UPV2024"
topic_destino = "sim/working/palet2"

# 2. Conexión rápida
mqttc = mqtt.Client(mqtt.CallbackAPIVersion.VERSION2)
#mqttc.username_pw_set(username=user, password=passwd)
mqttc.connect(broker, port, 60)

# 3. ¡Disparar el mensaje!
mensaje = "off"
mqttc.publish(topic_destino, mensaje)

# 4. Desconectar (Es buena práctica si el script termina aquí)
mqttc.disconnect()

--- Python program BorradoAzulejos ---
import time
from robodk import robolink    # RoboDK API
RDK = robolink.Robolink()


frame1 = RDK.Item('CintaCaja1')
frame2 = RDK.Item('CintaCaja2')
frame3 = RDK.Item('SMC ZXP7A01-ZP20U-X1 Vacuum Gripper')
lista_caja1 = frame1.Childs()
lista_caja2 = frame2.Childs()
lista_caja3 = frame3.Childs()

for item in lista_caja1:
    if item.Name().startswith('Azulejo'):
        item.Delete()

for item in lista_caja2:
    if item.Name().startswith('Azulejo'):
        item.Delete()

for item in lista_caja3:
    if item.Name().startswith('Azulejo'):
        item.Delete()
